{attribute addProperty BoxType "EL3102-0000-0016"}
{attribute addProperty Id "AI_Standard_ChannelAT %I*ARRAY[0..1] OF AI_Standard_Channel_8749C23514818.50WcStateAT %I*WcState_F855686C1620InfoDataAT %I*InfoData_BC63D37F80100"}
{attribute addProperty CRC "3770428868"}
{attribute addProperty SizeInBites "244"}
{attribute addProperty SizeInBytes "30.5"}
TYPE EL3102_8E42B51D :
STRUCT
	{attribute addProperty Name "AI_Standard_Channel"}
	AI_Standard_Channel : ARRAY[0..1] OF AI_Standard_Channel_8749C235;
	{attribute addProperty Name "WcState"}
	WcState : WcState_F855686C;
	{attribute addProperty Name "InfoData"}
	InfoData : InfoData_BC63D37F;
END_STRUCT
END_TYPE

(* stored: Version 1.2.0.0, ProductVersion 3.1.4024.9
   DUT EL3102_8E42B51D: Id {30bc07bc-6766-4a5a-abb2-997cc5a199ce} *)
